Universal Robots PolyScope program: sequential_full.urp

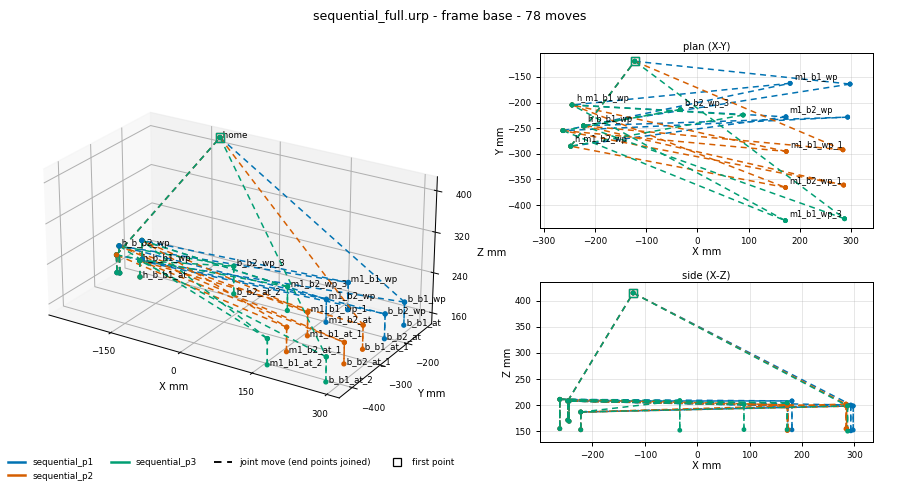
[picture p0: tool path of sequential_full.urp in frame base, 78 of 78 moves have a stored position in this frame; points joined in program order, loops and branches not executed]
Program sequential_full (installation=default directory=/programs/ITER createdIn=5.3.1.64192 lastSavedIn=5.3.1.64192 robotSerialNumber=20195300365)
Calibrated DH parameters: a=[-0.000093, -0.190649, -0.212673, 0.000091, -0.000205, 0]; d=[0.151591, 44.061648, -42.488068, -1.442789, 0.085322, 0.091911]; alpha=[1.570082, -0.003447, 0.007513, 1.572293, -1.571904, 0]; deltaTheta=[0, -0.672656, 0.728185, -0.055522, 0.000005, 0]
Robot Program (runOnlyOnce=true)
  Call sequential_p1
  Popup Message (haltProgram=false message=interaction inputType=Text)
  Call sequential_p2
  Popup Message (haltProgram=false message=interaction inputType=Text)
  Call sequential_p3
SubProgram -> sequential_p3
SubProgram -> sequential_p2
SubProgram -> sequential_p1
SubProgram sequential_p1 (keepSynchronizedWithDisk=true trackProgramExecution=false) programFile=/programs/ITER/sequential_p1.urp
  URCap Gripper Activate (Robotiq_Grippers, Robotiq Inc.) dataModel(ResetAndActivateKey=false)
  URCap Gripper (Robotiq_Grippers, Robotiq Inc.) dataModel(position=50.0, force=100.0, speed=100.0, positionInDouble=50.0, forceInDouble=100.0, speedInDouble=100.0, slaveIds=[9], blocking=true)
  MoveJ speed 60 deg/s, acceleration 80 deg/s^2 (useActiveTCP=true) feature=Base
    Waypoint home: TCP in base x=-122.15 y=-119.32 z=414.454 mm, rx=2.2563 ry=2.1459 rz=-0.0481 rad; joints [-85.681, -56.776, -79.802, -131.025, 89.944, -262.833] deg
  Folder Base
    MoveJ speed 60 deg/s, acceleration 80 deg/s^2 (useActiveTCP=true) feature=Base
      Waypoint b_b1_wp: TCP in base x=297.989 y=-163.874 z=198.695 mm, rx=2.2416 ry=2.1933 rz=-0.0875 rad; joints [-5.657, -99.775, -108.03, -64.017, 87.69, -183.98] deg
      Waypoint b_b1_at: TCP in base x=297.98 y=-163.89 z=152.63 mm, rx=2.2418 ry=2.1932 rz=-0.0874 rad; joints [-5.678, -106.278, -114.473, -51.073, 87.63, -183.927] deg
      URCap Gripper (Robotiq_Grippers, Robotiq Inc.) dataModel(position=100.0, force=100.0, speed=100.0, positionInDouble=100.0, forceInDouble=100.0, speedInDouble=100.0, slaveIds=[9], blocking=true)
      Waypoint b_b1_wp: TCP in base x=297.989 y=-163.874 z=198.695 mm, rx=2.2416 ry=2.1933 rz=-0.0875 rad; joints [-5.657, -99.775, -108.03, -64.017, 87.69, -183.98] deg
      Waypoint h_b_b1_wp: TCP in base x=-222.187 y=-245.349 z=187.06 mm, rx=-3.1315 ry=0.0204 rz=0.0123 rad; joints [-108.957, -99.116, -113.081, -58.146, 89.665, -197.782] deg
      Waypoint h_b_b1_at: TCP in base x=-222.188 y=-245.348 z=153.24 mm, rx=-3.1314 ry=0.0204 rz=0.0122 rad; joints [-108.969, -104.391, -117.643, -48.312, 89.612, -197.745] deg
      URCap Gripper (Robotiq_Grippers, Robotiq Inc.) dataModel(position=50.0, force=100.0, speed=100.0, positionInDouble=50.0, forceInDouble=100.0, speedInDouble=100.0, slaveIds=[9], blocking=true)
      Waypoint h_b_b1_wp: TCP in base x=-222.187 y=-245.349 z=187.06 mm, rx=-3.1315 ry=0.0204 rz=0.0123 rad; joints [-108.957, -99.116, -113.081, -58.146, 89.665, -197.782] deg
    MoveJ speed 60 deg/s, acceleration 80 deg/s^2 (useActiveTCP=true) feature=Base
      Waypoint b_b2_wp: TCP in base x=293.357 y=-228.364 z=200.348 mm, rx=2.2516 ry=2.1757 rz=-0.0473 rad; joints [-17.02, -106.79, -99.111, -64.372, 88.479, -194.689] deg
      Waypoint b_b2_at: TCP in base x=293.371 y=-228.346 z=151.163 mm, rx=2.2516 ry=2.1757 rz=-0.0473 rad; joints [-17.033, -113.072, -105.562, -51.642, 88.423, -194.639] deg
      URCap Gripper (Robotiq_Grippers, Robotiq Inc.) dataModel(position=100.0, force=100.0, speed=100.0, positionInDouble=100.0, forceInDouble=100.0, speedInDouble=100.0, slaveIds=[9], blocking=true)
      Waypoint b_b2_wp: TCP in base x=293.357 y=-228.364 z=200.348 mm, rx=2.2516 ry=2.1757 rz=-0.0473 rad; joints [-17.02, -106.79, -99.111, -64.372, 88.479, -194.689] deg
      Waypoint h_b_b2_wp: TCP in base x=-262.196 y=-254.726 z=211.351 mm, rx=-3.0605 ry=0.0443 rz=-0.0223 rad; joints [-114.749, -105.359, -96.042, -73.109, 89.199, -202.734] deg
      Waypoint h_b_b2_at: TCP in base x=-262.208 y=-254.718 z=155.33 mm, rx=-3.0605 ry=0.0443 rz=-0.0223 rad; joints [-114.774, -111.736, -104.192, -58.581, 89.146, -202.674] deg
      URCap Gripper (Robotiq_Grippers, Robotiq Inc.) dataModel(position=50.0, force=100.0, speed=100.0, positionInDouble=50.0, forceInDouble=100.0, speedInDouble=100.0, slaveIds=[9], blocking=true)
      Waypoint h_b_b2_wp: TCP in base x=-262.196 y=-254.726 z=211.351 mm, rx=-3.0605 ry=0.0443 rz=-0.0223 rad; joints [-114.749, -105.359, -96.042, -73.109, 89.199, -202.734] deg
  Folder Mid_1
    MoveJ speed 60 deg/s, acceleration 80 deg/s^2 (useActiveTCP=true) feature=Base
      Waypoint m1_b1_wp: TCP in base x=181.055 y=-162.39 z=208.274 mm, rx=2.2824 ry=2.1481 rz=-0.0224 rad; joints [-9.334, -71.677, -131.429, -67.006, 89.476, -185.444] deg
      Waypoint m1_b1_at: TCP in base x=181.066 y=-162.388 z=153.109 mm, rx=2.2824 ry=2.1481 rz=-0.0224 rad; joints [-9.367, -82.083, -142.13, -45.899, 89.364, -185.356] deg
      URCap Gripper (Robotiq_Grippers, Robotiq Inc.) dataModel(position=100.0, force=100.0, speed=100.0, positionInDouble=100.0, forceInDouble=100.0, speedInDouble=100.0, slaveIds=[9], blocking=true)
      Waypoint m1_b1_wp: TCP in base x=181.055 y=-162.39 z=208.274 mm, rx=2.2824 ry=2.1481 rz=-0.0224 rad; joints [-9.334, -71.677, -131.429, -67.006, 89.476, -185.444] deg
      Waypoint h_m1_b1_wp: TCP in base x=-244.449 y=-204.582 z=208.1 mm, rx=2.2684 ry=2.1196 rz=0.0229 rad; joints [-116.825, -93.932, -112.747, -63.308, 92.582, -292.535] deg
      Waypoint h_m1_b1_at: TCP in base x=-244.447 y=-204.577 z=169.457 mm, rx=2.2685 ry=2.1196 rz=0.0229 rad; joints [-116.841, -99.299, -118.834, -51.852, 92.525, -292.487] deg
      URCap Gripper (Robotiq_Grippers, Robotiq Inc.) dataModel(position=50.0, force=100.0, speed=100.0, positionInDouble=50.0, forceInDouble=100.0, speedInDouble=100.0, slaveIds=[9], blocking=true)
      Waypoint h_m1_b1_wp: TCP in base x=-244.449 y=-204.582 z=208.1 mm, rx=2.2684 ry=2.1196 rz=0.0229 rad; joints [-116.825, -93.932, -112.747, -63.308, 92.582, -292.535] deg
    MoveJ speed 60 deg/s, acceleration 80 deg/s^2 (useActiveTCP=true) feature=Base
      Waypoint m1_b2_wp: TCP in base x=172.9 y=-227.784 z=198.59 mm, rx=2.2733 ry=2.1297 rz=0.0128 rad; joints [-25.861, -85.885, -124.428, -58.034, 90.195, -201.672] deg
      Waypoint m1_b2_at: TCP in base x=172.893 y=-227.779 z=152.722 mm, rx=2.2733 ry=2.1297 rz=0.0127 rad; joints [-25.879, -94.277, -131.683, -42.391, 90.103, -201.614] deg
      URCap Gripper (Robotiq_Grippers, Robotiq Inc.) dataModel(position=100.0, force=100.0, speed=100.0, positionInDouble=100.0, forceInDouble=100.0, speedInDouble=100.0, slaveIds=[9], blocking=true)
      Waypoint m1_b2_wp: TCP in base x=172.9 y=-227.784 z=198.59 mm, rx=2.2733 ry=2.1297 rz=0.0128 rad; joints [-25.861, -85.885, -124.428, -58.034, 90.195, -201.672] deg
      Waypoint h_m1_b2_wp: TCP in base x=-247.009 y=-285.144 z=208.116 mm, rx=2.2684 ry=2.1195 rz=0.0229 rad; joints [-111.389, -107.719, -95.772, -66.28, 92.556, -287.152] deg
      Waypoint h_m1_b2_at: TCP in base x=-246.994 y=-285.166 z=171.647 mm, rx=2.2684 ry=2.1196 rz=0.0229 rad; joints [-111.399, -111.783, -101.037, -56.949, 92.516, -287.113] deg
      URCap Gripper (Robotiq_Grippers, Robotiq Inc.) dataModel(position=50.0, force=100.0, speed=100.0, positionInDouble=50.0, forceInDouble=100.0, speedInDouble=100.0, slaveIds=[9], blocking=true)
      Waypoint h_m1_b2_wp: TCP in base x=-247.009 y=-285.144 z=208.116 mm, rx=2.2684 ry=2.1195 rz=0.0229 rad; joints [-111.389, -107.719, -95.772, -66.28, 92.556, -287.152] deg
  MoveJ speed 60 deg/s, acceleration 80 deg/s^2 (useActiveTCP=true) feature=Base
    Waypoint home: TCP in base x=-122.15 y=-119.32 z=414.454 mm, rx=2.2563 ry=2.1459 rz=-0.0481 rad; joints [-85.681, -56.776, -79.802, -131.025, 89.944, -262.833] deg
SubProgram sequential_p2 (keepSynchronizedWithDisk=true trackProgramExecution=false) programFile=/programs/ITER/sequential_p2.urp
  URCap Gripper Activate (Robotiq_Grippers, Robotiq Inc.) dataModel(ResetAndActivateKey=false)
  URCap Gripper (Robotiq_Grippers, Robotiq Inc.) dataModel(position=50.0, force=100.0, speed=100.0, positionInDouble=50.0, forceInDouble=100.0, speedInDouble=100.0, slaveIds=[9], blocking=true)
  MoveJ speed 60 deg/s, acceleration 80 deg/s^2 (useActiveTCP=true) feature=Base
    Waypoint home: TCP in base x=-122.15 y=-119.32 z=414.454 mm, rx=2.2563 ry=2.1459 rz=-0.0481 rad; joints [-85.681, -56.776, -79.802, -131.025, 89.944, -262.833] deg
  Folder Base
    MoveJ speed 60 deg/s, acceleration 80 deg/s^2 (useActiveTCP=true) feature=Base
      Waypoint b_b1_wp_1: TCP in base x=284.13 y=-292.134 z=202.324 mm, rx=2.2344 ry=2.1191 rz=-0.0341 rad; joints [-26.664, -114.085, -89.487, -63.473, 87.858, -203.352] deg
      Waypoint b_b1_at_1: TCP in base x=284.119 y=-292.135 z=154.941 mm, rx=2.2346 ry=2.1191 rz=-0.0343 rad; joints [-26.679, -119.503, -95.459, -52.092, 87.809, -203.308] deg
      URCap Gripper (Robotiq_Grippers, Robotiq Inc.) dataModel(position=100.0, force=100.0, speed=100.0, positionInDouble=100.0, forceInDouble=100.0, speedInDouble=100.0, slaveIds=[9], blocking=true)
      Waypoint b_b1_wp_2: TCP in base x=284.13 y=-292.134 z=202.324 mm, rx=2.2344 ry=2.1191 rz=-0.0341 rad; joints [-26.664, -114.085, -89.487, -63.473, 87.858, -203.352] deg
      Waypoint h_b_b1_wp: TCP in base x=-222.187 y=-245.349 z=187.06 mm, rx=-3.1315 ry=0.0204 rz=0.0123 rad; joints [-108.957, -99.116, -113.081, -58.146, 89.665, -197.782] deg
      Waypoint h_b_b1_at: TCP in base x=-222.188 y=-245.348 z=153.24 mm, rx=-3.1314 ry=0.0204 rz=0.0122 rad; joints [-108.969, -104.391, -117.643, -48.312, 89.612, -197.745] deg
      URCap Gripper (Robotiq_Grippers, Robotiq Inc.) dataModel(position=50.0, force=100.0, speed=100.0, positionInDouble=50.0, forceInDouble=100.0, speedInDouble=100.0, slaveIds=[9], blocking=true)
      Waypoint h_b_b1_wp: TCP in base x=-222.187 y=-245.349 z=187.06 mm, rx=-3.1315 ry=0.0204 rz=0.0123 rad; joints [-108.957, -99.116, -113.081, -58.146, 89.665, -197.782] deg
    MoveJ speed 60 deg/s, acceleration 80 deg/s^2 (useActiveTCP=true) feature=Base
      Waypoint b_b2_wp_1: TCP in base x=285.472 y=-360.969 z=198.014 mm, rx=2.2366 ry=2.1589 rz=-0.0532 rad; joints [-34.767, -127.303, -68.664, -72.529, 87.977, -212.535] deg
      Waypoint b_b2_at_1: TCP in base x=285.465 y=-360.98 z=156.253 mm, rx=2.2366 ry=2.1588 rz=-0.0532 rad; joints [-34.783, -130.917, -74.259, -63.319, 87.955, -212.495] deg
      URCap Gripper (Robotiq_Grippers, Robotiq Inc.) dataModel(position=100.0, force=100.0, speed=100.0, positionInDouble=100.0, forceInDouble=100.0, speedInDouble=100.0, slaveIds=[9], blocking=true)
      Waypoint b_b2_wp_2: TCP in base x=285.472 y=-360.969 z=198.014 mm, rx=2.2366 ry=2.1589 rz=-0.0532 rad; joints [-34.767, -127.303, -68.664, -72.529, 87.977, -212.535] deg
      Waypoint h_b_b2_wp: TCP in base x=-262.196 y=-254.726 z=211.351 mm, rx=-3.0605 ry=0.0443 rz=-0.0223 rad; joints [-114.749, -105.359, -96.042, -73.109, 89.199, -202.734] deg
      Waypoint h_b_b2_at: TCP in base x=-262.208 y=-254.718 z=155.33 mm, rx=-3.0605 ry=0.0443 rz=-0.0223 rad; joints [-114.774, -111.736, -104.192, -58.581, 89.146, -202.674] deg
      URCap Gripper (Robotiq_Grippers, Robotiq Inc.) dataModel(position=50.0, force=100.0, speed=100.0, positionInDouble=50.0, forceInDouble=100.0, speedInDouble=100.0, slaveIds=[9], blocking=true)
      Waypoint h_b_b2_wp: TCP in base x=-262.196 y=-254.726 z=211.351 mm, rx=-3.0605 ry=0.0443 rz=-0.0223 rad; joints [-114.749, -105.359, -96.042, -73.109, 89.199, -202.734] deg
  Folder Mid_1
    MoveJ speed 60 deg/s, acceleration 80 deg/s^2 (useActiveTCP=true) feature=Base
      Waypoint m1_b1_wp_1: TCP in base x=173.538 y=-295.326 z=200.585 mm, rx=2.2061 ry=2.2228 rz=-0.0106 rad; joints [-37.214, -100.014, -108.204, -61.217, 89.822, -217.247] deg
      Waypoint m1_b1_at_1: TCP in base x=173.554 y=-295.318 z=153.797 mm, rx=2.2061 ry=2.223 rz=-0.0106 rad; joints [-37.227, -106.714, -114.649, -48.075, 89.755, -217.198] deg
      URCap Gripper (Robotiq_Grippers, Robotiq Inc.) dataModel(position=100.0, force=100.0, speed=100.0, positionInDouble=100.0, forceInDouble=100.0, speedInDouble=100.0, slaveIds=[9], blocking=true)
      Waypoint m1_b1_wp_2: TCP in base x=173.538 y=-295.326 z=200.585 mm, rx=2.2061 ry=2.2228 rz=-0.0106 rad; joints [-37.214, -100.014, -108.204, -61.217, 89.822, -217.247] deg
      Waypoint h_m1_b1_wp: TCP in base x=-244.449 y=-204.582 z=208.1 mm, rx=2.2684 ry=2.1196 rz=0.0229 rad; joints [-116.825, -93.932, -112.747, -63.308, 92.582, -292.535] deg
      Waypoint h_m1_b1_at: TCP in base x=-244.447 y=-204.577 z=169.457 mm, rx=2.2685 ry=2.1196 rz=0.0229 rad; joints [-116.841, -99.299, -118.834, -51.852, 92.525, -292.487] deg
      URCap Gripper (Robotiq_Grippers, Robotiq Inc.) dataModel(position=50.0, force=100.0, speed=100.0, positionInDouble=50.0, forceInDouble=100.0, speedInDouble=100.0, slaveIds=[9], blocking=true)
      Waypoint h_m1_b1_wp: TCP in base x=-244.449 y=-204.582 z=208.1 mm, rx=2.2684 ry=2.1196 rz=0.0229 rad; joints [-116.825, -93.932, -112.747, -63.308, 92.582, -292.535] deg
    MoveJ speed 60 deg/s, acceleration 80 deg/s^2 (useActiveTCP=true) feature=Base
      Waypoint m1_b2_wp_1: TCP in base x=172.109 y=-365.692 z=199.867 mm, rx=2.2648 ry=2.1714 rz=0.0103 rad; joints [-46.162, -114.393, -88.528, -66.782, 90.646, -223.425] deg
      Waypoint m1_b2_at_1: TCP in base x=172.105 y=-365.689 z=151.683 mm, rx=2.2649 ry=2.1715 rz=0.0104 rad; joints [-46.178, -119.803, -94.665, -55.241, 90.602, -223.381] deg
      URCap Gripper (Robotiq_Grippers, Robotiq Inc.) dataModel(position=100.0, force=100.0, speed=100.0, positionInDouble=100.0, forceInDouble=100.0, speedInDouble=100.0, slaveIds=[9], blocking=true)
      Waypoint m1_b2_wp_2: TCP in base x=172.109 y=-365.692 z=199.867 mm, rx=2.2648 ry=2.1714 rz=0.0103 rad; joints [-46.162, -114.393, -88.528, -66.782, 90.646, -223.425] deg
      Waypoint h_m1_b2_wp: TCP in base x=-247.009 y=-285.144 z=208.116 mm, rx=2.2684 ry=2.1195 rz=0.0229 rad; joints [-111.389, -107.719, -95.772, -66.28, 92.556, -287.152] deg
      Waypoint h_m1_b2_at: TCP in base x=-246.994 y=-285.166 z=171.647 mm, rx=2.2684 ry=2.1196 rz=0.0229 rad; joints [-111.399, -111.783, -101.037, -56.949, 92.516, -287.113] deg
      URCap Gripper (Robotiq_Grippers, Robotiq Inc.) dataModel(position=50.0, force=100.0, speed=100.0, positionInDouble=50.0, forceInDouble=100.0, speedInDouble=100.0, slaveIds=[9], blocking=true)
      Waypoint h_m1_b2_wp: TCP in base x=-247.009 y=-285.144 z=208.116 mm, rx=2.2684 ry=2.1195 rz=0.0229 rad; joints [-111.389, -107.719, -95.772, -66.28, 92.556, -287.152] deg
  MoveJ speed 60 deg/s, acceleration 80 deg/s^2 (useActiveTCP=true) feature=Base
    Waypoint home: TCP in base x=-122.15 y=-119.32 z=414.454 mm, rx=2.2563 ry=2.1459 rz=-0.0481 rad; joints [-85.681, -56.776, -79.802, -131.025, 89.944, -262.833] deg
SubProgram sequential_p3 (keepSynchronizedWithDisk=true trackProgramExecution=false) programFile=/programs/ITER/sequential_p3.urp
  URCap Gripper Activate (Robotiq_Grippers, Robotiq Inc.) dataModel(ResetAndActivateKey=false)
  URCap Gripper (Robotiq_Grippers, Robotiq Inc.) dataModel(position=50.0, force=100.0, speed=100.0, positionInDouble=50.0, forceInDouble=100.0, speedInDouble=100.0, slaveIds=[9], blocking=true)
  MoveJ speed 60 deg/s, acceleration 80 deg/s^2 (useActiveTCP=true) feature=Base
    Waypoint home: TCP in base x=-122.15 y=-119.32 z=414.454 mm, rx=2.2563 ry=2.1459 rz=-0.0481 rad; joints [-85.681, -56.776, -79.802, -131.025, 89.944, -262.833] deg
  Folder Base
    MoveJ speed 60 deg/s, acceleration 80 deg/s^2 (useActiveTCP=true) feature=Base
      Waypoint b_b1_wp_3: TCP in base x=287.27 y=-426.687 z=198.703 mm, rx=2.2572 ry=2.1295 rz=-0.0633 rad; joints [-40.865, -143.306, -39.499, -85.215, 87.731, -217.488] deg
      Waypoint b_b1_at_2: TCP in base x=287.269 y=-426.683 z=150.489 mm, rx=2.2571 ry=2.1295 rz=-0.0633 rad; joints [-40.886, -145.62, -48.126, -74.275, 87.723, -217.437] deg
      URCap Gripper (Robotiq_Grippers, Robotiq Inc.) dataModel(position=100.0, force=100.0, speed=100.0, positionInDouble=100.0, forceInDouble=100.0, speedInDouble=100.0, slaveIds=[9], blocking=true)
      Waypoint b_b1_wp_4: TCP in base x=287.27 y=-426.687 z=198.703 mm, rx=2.2572 ry=2.1295 rz=-0.0633 rad; joints [-40.865, -143.306, -39.499, -85.215, 87.731, -217.488] deg
      Waypoint h_b_b1_wp: TCP in base x=-222.187 y=-245.349 z=187.06 mm, rx=-3.1315 ry=0.0204 rz=0.0123 rad; joints [-108.957, -99.116, -113.081, -58.146, 89.665, -197.782] deg
      Waypoint h_b_b1_at: TCP in base x=-222.188 y=-245.348 z=153.24 mm, rx=-3.1314 ry=0.0204 rz=0.0122 rad; joints [-108.969, -104.391, -117.643, -48.312, 89.612, -197.745] deg
      URCap Gripper (Robotiq_Grippers, Robotiq Inc.) dataModel(position=50.0, force=100.0, speed=100.0, positionInDouble=50.0, forceInDouble=100.0, speedInDouble=100.0, slaveIds=[9], blocking=true)
      Waypoint h_b_b1_wp: TCP in base x=-222.187 y=-245.349 z=187.06 mm, rx=-3.1315 ry=0.0204 rz=0.0123 rad; joints [-108.957, -99.116, -113.081, -58.146, 89.665, -197.782] deg
    MoveJ speed 60 deg/s, acceleration 80 deg/s^2 (useActiveTCP=true) feature=Base
      Waypoint b_b2_wp_3: TCP in base x=-33.1 y=-213.495 z=208.789 mm, rx=2.2331 ry=2.1669 rz=-0.0323 rad; joints [-61.64, -60.837, -137.744, -69.392, 89.733, -239.518] deg
      Waypoint b_b2_at_2: TCP in base x=-33.102 y=-213.489 z=152.337 mm, rx=2.2331 ry=2.167 rz=-0.0323 rad; joints [-61.683, -72.125, -150.112, -45.739, 89.609, -239.421] deg
      URCap Gripper (Robotiq_Grippers, Robotiq Inc.) dataModel(position=100.0, force=100.0, speed=100.0, positionInDouble=100.0, forceInDouble=100.0, speedInDouble=100.0, slaveIds=[9], blocking=true)
      Waypoint b_b2_wp_4: TCP in base x=-33.1 y=-213.495 z=208.789 mm, rx=2.2331 ry=2.1669 rz=-0.0323 rad; joints [-61.64, -60.837, -137.744, -69.392, 89.733, -239.518] deg
      Waypoint h_b_b2_wp: TCP in base x=-262.196 y=-254.726 z=211.351 mm, rx=-3.0605 ry=0.0443 rz=-0.0223 rad; joints [-114.749, -105.359, -96.042, -73.109, 89.199, -202.734] deg
      Waypoint h_b_b2_at: TCP in base x=-262.208 y=-254.718 z=155.33 mm, rx=-3.0605 ry=0.0443 rz=-0.0223 rad; joints [-114.774, -111.736, -104.192, -58.581, 89.146, -202.674] deg
      URCap Gripper (Robotiq_Grippers, Robotiq Inc.) dataModel(position=50.0, force=100.0, speed=100.0, positionInDouble=50.0, forceInDouble=100.0, speedInDouble=100.0, slaveIds=[9], blocking=true)
      Waypoint h_b_b2_wp: TCP in base x=-262.196 y=-254.726 z=211.351 mm, rx=-3.0605 ry=0.0443 rz=-0.0223 rad; joints [-114.749, -105.359, -96.042, -73.109, 89.199, -202.734] deg
  Folder Mid_1
    MoveJ speed 60 deg/s, acceleration 80 deg/s^2 (useActiveTCP=true) feature=Base
      Waypoint m1_b1_wp_3: TCP in base x=171.816 y=-430.356 z=204.684 mm, rx=2.26 ry=2.1667 rz=-0.0282 rad; joints [-51.724, -128.073, -65.156, -76.01, 89.303, -229.106] deg
      Waypoint m1_b1_at_2: TCP in base x=171.786 y=-430.365 z=153.694 mm, rx=2.2601 ry=2.1667 rz=-0.0282 rad; joints [-51.746, -132.202, -72.305, -64.735, 89.276, -229.058] deg
      URCap Gripper (Robotiq_Grippers, Robotiq Inc.) dataModel(position=100.0, force=100.0, speed=100.0, positionInDouble=100.0, forceInDouble=100.0, speedInDouble=100.0, slaveIds=[9], blocking=true)
      Waypoint m1_b1_wp_4: TCP in base x=171.816 y=-430.356 z=204.684 mm, rx=2.26 ry=2.1667 rz=-0.0282 rad; joints [-51.724, -128.073, -65.156, -76.01, 89.303, -229.106] deg
      Waypoint h_m1_b1_wp: TCP in base x=-244.449 y=-204.582 z=208.1 mm, rx=2.2684 ry=2.1196 rz=0.0229 rad; joints [-116.825, -93.932, -112.747, -63.308, 92.582, -292.535] deg
      Waypoint h_m1_b1_at: TCP in base x=-244.447 y=-204.577 z=169.457 mm, rx=2.2685 ry=2.1196 rz=0.0229 rad; joints [-116.841, -99.299, -118.834, -51.852, 92.525, -292.487] deg
      URCap Gripper (Robotiq_Grippers, Robotiq Inc.) dataModel(position=50.0, force=100.0, speed=100.0, positionInDouble=50.0, forceInDouble=100.0, speedInDouble=100.0, slaveIds=[9], blocking=true)
      Waypoint h_m1_b1_wp: TCP in base x=-244.449 y=-204.582 z=208.1 mm, rx=2.2684 ry=2.1196 rz=0.0229 rad; joints [-116.825, -93.932, -112.747, -63.308, 92.582, -292.535] deg
    MoveJ speed 60 deg/s, acceleration 80 deg/s^2 (useActiveTCP=true) feature=Base
      Waypoint m1_b2_wp_3: TCP in base x=89.366 y=-224.31 z=201.565 mm, rx=-2.2386 ry=-2.1806 rz=-0.0102 rad; joints [-36.103, -72.547, -132.567, -65.683, 90.9, -214.176] deg
      Waypoint m1_b2_at_2: TCP in base x=89.368 y=-224.313 z=153.584 mm, rx=-2.2387 ry=-2.1806 rz=-0.0101 rad; joints [-36.132, -81.828, -141.776, -47.193, 90.798, -214.098] deg
      URCap Gripper (Robotiq_Grippers, Robotiq Inc.) dataModel(position=100.0, force=100.0, speed=100.0, positionInDouble=100.0, forceInDouble=100.0, speedInDouble=100.0, slaveIds=[9], blocking=true)
      Waypoint m1_b2_wp_4: TCP in base x=89.366 y=-224.31 z=201.565 mm, rx=-2.2386 ry=-2.1806 rz=-0.0102 rad; joints [-36.103, -72.547, -132.567, -65.683, 90.9, -214.176] deg
      Waypoint h_m1_b2_wp: TCP in base x=-247.009 y=-285.144 z=208.116 mm, rx=2.2684 ry=2.1195 rz=0.0229 rad; joints [-111.389, -107.719, -95.772, -66.28, 92.556, -287.152] deg
      Waypoint h_m1_b2_at: TCP in base x=-246.994 y=-285.166 z=171.647 mm, rx=2.2684 ry=2.1196 rz=0.0229 rad; joints [-111.399, -111.783, -101.037, -56.949, 92.516, -287.113] deg
      URCap Gripper (Robotiq_Grippers, Robotiq Inc.) dataModel(position=50.0, force=100.0, speed=100.0, positionInDouble=50.0, forceInDouble=100.0, speedInDouble=100.0, slaveIds=[9], blocking=true)
      Waypoint h_m1_b2_wp: TCP in base x=-247.009 y=-285.144 z=208.116 mm, rx=2.2684 ry=2.1195 rz=0.0229 rad; joints [-111.389, -107.719, -95.772, -66.28, 92.556, -287.152] deg
  MoveJ speed 60 deg/s, acceleration 80 deg/s^2 (useActiveTCP=true) feature=Base
    Waypoint home: TCP in base x=-122.15 y=-119.32 z=414.454 mm, rx=2.2563 ry=2.1459 rz=-0.0481 rad; joints [-85.681, -56.776, -79.802, -131.025, 89.944, -262.833] deg
